// Mitsubishi GX Works2 project: BSFL   PLC: Q03UDV

PROGRAM MAIN
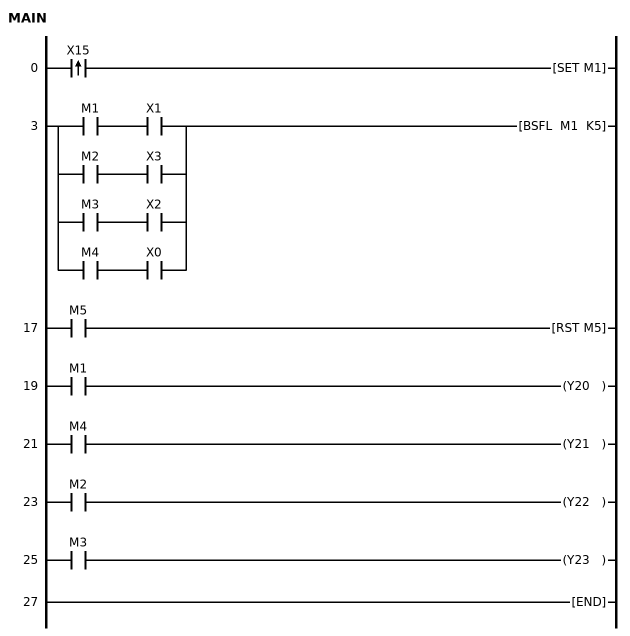
0     LDP     X15
      SET     M1
3     LD      M1
      AND     X1
      LD      M2
      AND     X3
      ORB
      LD      M3
      AND     X2
      ORB
      LD      M4
      AND     X0
      ORB
      BSFL    M1 K5
17    LD      M5
      RST     M5
19    LD      M1
      OUT     Y20
21    LD      M4
      OUT     Y21
23    LD      M2
      OUT     Y22
25    LD      M3
      OUT     Y23
27    END
END_PROGRAM
